TYPE ST_Parameters_1 :
STRUCT
	fCyclicTime : LREAL := 0.01; 
	stAnimationScaling : ST_AnimationScaling;
	stPistonRange : ST_PistonRange; 
	stCraneKinematics : ST_CraneKinematics;
END_STRUCT
END_TYPE

(* stored: Version 1.1.0.1, ProductVersion 3.1.4024.9
   DUT ST_Parameters_1: Id {327f9d83-5c16-4c45-a49f-a5c776ff898b} *)
